(* IEC 61131-3 sources: volt/packages/volt-lsp-iec/test-corpus/awa-palletizer/Device/Plc Logic/Application/Library Manager/CmpErrors, 2 files *)

(* ---- ERRORS.gvl ---- *)
VAR_GLOBAL
	ERR_OK : UDINT := 16#0;
	ERR_FAILED : UDINT := 16#1;
	ERR_PARAMETER : UDINT := 16#2;
	ERR_NOTINITIALIZED : UDINT := 16#3;
	ERR_VERSION : UDINT := 16#4;
	ERR_TIMEOUT : UDINT := 16#5;
	ERR_NOBUFFER : UDINT := 16#6;
	ERR_PENDING : UDINT := 16#A;
	ERR_NUMPENDING : UDINT := 16#B;
	ERR_NOTIMPLEMENTED : UDINT := 16#C;
	ERR_INVALIDID : UDINT := 16#D;
	ERR_OVERFLOW : UDINT := 16#E;
	ERR_BUFFERSIZE : UDINT := 16#F;
	ERR_NO_OBJECT : UDINT := 16#10;
	ERR_NOMEMORY : UDINT := 16#11;
	ERR_DUPLICATE : UDINT := 16#12;
	ERR_MEMORY_OVERWRITE : UDINT := 16#13;
	ERR_INVALID_HANDLE : UDINT := 16#14;
	ERR_END_OF_OBJECT : UDINT := 16#15;
	ERR_NO_CHANGE : UDINT := 16#16;
	ERR_INVALID_INTERFACE : UDINT := 16#17;
	ERR_NOT_SUPPORTED : UDINT := 16#18;
	ERR_NO_ACCESS_RIGHTS : UDINT := 16#19;
	ERR_OUT_OF_LIMITS : UDINT := 16#1A;
	ERR_ENTRIES_REMAINING : UDINT := 16#1B;
	ERR_INVALID_SESSION_ID : UDINT := 16#1C;
	ERR_EXCEPTION : UDINT := 16#1D;
	ERR_SOCK_NOTINITIALIZED : UDINT := 16#201;
	ERR_SOCK_NOTSOCKET : UDINT := 16#202;
	ERR_SOCK_AFUNSUPPORTED : UDINT := 16#203;
	ERR_SOCK_PROTOUNSUPPORTED : UDINT := 16#204;
	ERR_SOCK_NOBUFFER : UDINT := 16#205;
	ERR_SOCK_WOULDBLOCK : UDINT := 16#206;
	ERR_SOCK_ADDRINUSE : UDINT := 16#207;
	ERR_SOCK_ADDRNOTAVAILABLE : UDINT := 16#208;
	ERR_SOCK_CONNREFUSED : UDINT := 16#209;
	ERR_SOCK_TIMEDOUT : UDINT := 16#20A;
	ERR_SOCK_HOSTNOTFOUND : UDINT := 16#20B;
	ERR_SOCK_HOSTUNREACHABLE : UDINT := 16#20C;
	ERR_SOCK_ISCONNECTED : UDINT := 16#20D;
	ERR_SOCK_NOTCONNECTED : UDINT := 16#20E;
	ERR_SOCK_SHUTDOWN : UDINT := 16#20F;
	ERR_SOCK_MSGSIZE : UDINT := 16#210;
	ERR_SOCK_CLOSED : UDINT := 16#211;
END_VAR

(* ---- HANDLEERRORS.gvl ---- *)
VAR_GLOBAL
	RTS_INVALID_HANDLE : RTS_IEC_HANDLE := SINT_TO_DWORD(-1);
END_VAR
